PROGRAM UpperPreserDrive
VAR
	fbUupperPreser: FB_RevMotorControl;
	
	bStop: BOOL;
	
END_VAR

fbUupperPreser(
	bForward:=.bTopPreserCmdDown , 
	bReverse:=.bTopPreserCmdUp , 
	bStop:=bStop , 
	bThermalOk:=.bTopPreserMotorOk , 
	bLimitSwitchFwd:=TRUE , 
	bLimitSwitchRev:=.bTopPreserClosed , 
	bEmergencyStop:=.bEstopOk , 
	bEnable:=bControlOn , 
	bRunForward=>.bTopPreserDown , 
	bRunReverse=>.bTopPreserUp , 
	bRunning=> , 
	bFault=> , 
	bReady=> );

END_PROGRAM

(* stored: Version 1.1.0.1, ProductVersion 3.1.4024.15
   POU UpperPreserDrive: Id {7039e87a-c5a8-4af5-aaec-fe52d9ca3e28}, SpecialFunc None *)
